INTERFACE PUBLIC UnsuspendingCommands EXTENDS RunningStateCommands, ActionStateCommands, HoldableStateCommands

END_INTERFACE

(* stored: Version 1.1.0.1, ProductVersion 3.1.4026.18
   Itf UnsuspendingCommands: Id {100e6468-f259-0ece-08ab-ed447511f482} *)
